INTERFACE IStreamReader

METHOD Read_BLOB
VAR_INPUT
    Value : ANY;
END_VAR
END_METHOD

METHOD Read_BOOL : BOOL;
END_METHOD

METHOD Read_BYTE : BYTE;
END_METHOD

METHOD Read_DINT : DINT;
END_METHOD

METHOD Read_INT : INT;
END_METHOD

METHOD Read_LINT : LINT;
END_METHOD

METHOD Read_LREAL : LREAL;
END_METHOD

METHOD Read_PVOID : PVOID;
END_METHOD

METHOD Read_REAL : REAL;
END_METHOD

METHOD Read_STRING : STRING(255);
END_METHOD

METHOD Read_UDINT : UDINT;
END_METHOD

METHOD Read_UINT : UINT;
END_METHOD

METHOD Read_ULINT : ULINT;
END_METHOD

METHOD Seek: IStreamWriter
VAR_INPUT
    Position : UDINT;
END_VAR
END_METHOD

END_INTERFACE

(* stored: Version 1.1.0.1, ProductVersion 3.1.4024.3
   Itf IStreamReader: Id {4ce154d4-15b3-0d46-1c83-b5e5fa9c119b}
   Folder Methods: Id {b8877614-48d5-0eca-2865-22e970702037}
   Method Read_BLOB: Id {f8c9a894-7e28-4c4d-9d66-adf775a9e61a}
   Method Read_BOOL: Id {e1bdd036-7870-0f43-0e36-b5bb859b7000}
   Method Read_BYTE: Id {3ccda0cd-8655-0f56-2bc9-c58e6daa3ce8}
   Method Read_DINT: Id {48ce2b84-3168-03ca-12f0-71cd392d8654}
   Method Read_INT: Id {0148bb1b-7254-009d-3f2a-34f63964ce35}
   Method Read_LINT: Id {6c195aa8-b80e-02db-1b75-c81ae8eff187}
   Method Read_LREAL: Id {759500c4-a674-0ff0-2e2d-d445694ce533}
   Method Read_PVOID: Id {3ebc800b-5c5f-0c00-00d9-41734ef2561d}
   Method Read_REAL: Id {76140bff-57d3-00c0-2b2c-0e5854607f62}
   Method Read_STRING: Id {b6f5d3cd-32d2-0aa1-36c6-26f76c20da1d}
   Method Read_UDINT: Id {bc95bb0c-f0ce-0a03-227c-c8ac3d307b3a}
   Method Read_UINT: Id {cda1de9e-731f-09c7-37ed-3632355d115f}
   Method Read_ULINT: Id {c0f7078d-b578-031e-227a-d5f3c9e4196b}
   Method Seek: Id {86b70d1c-7207-094c-05c9-c562e8f29569} *)
